(* IEC 61131-3 sources: MSMP/PLC_Station/Source/FB, 12 files *)

(* ---- FB_CANopenManager.st ---- *)
FUNCTION_BLOCK FB_CANopenManager
VAR_INPUT
 Enable:BOOL;
END_VAR
VAR_OUTPUT
 Ready:BOOL;
END_VAR
IF Enable THEN
 Ready:=TRUE;
ELSE
 Ready:=FALSE;
END_IF;
END_FUNCTION_BLOCK

(* ---- FB_ConnectionMonitor.st ---- *)
FUNCTION_BLOCK FB_ConnectionMonitor
VAR_INPUT Connected:BOOL; END_VAR
VAR_OUTPUT Alarm:BOOL; END_VAR
Alarm:=NOT Connected;
END_FUNCTION_BLOCK

(* ---- FB_DataAcquisition.st ---- *)
FUNCTION_BLOCK FB_DataAcquisition
VAR_INPUT
    Enable : BOOL;
END_VAR
VAR_OUTPUT
    Done : BOOL;
END_VAR

IF Enable THEN
    // TODO: Read 6 CANopen encoders
    Done := TRUE;
ELSE
    Done := FALSE;
END_IF;

END_FUNCTION_BLOCK

(* ---- FB_Diagnostics.st ---- *)
FUNCTION_BLOCK FB_Diagnostics
VAR_INPUT
 CAN_OK:BOOL;
 MODBUS_OK:BOOL;
END_VAR
VAR_OUTPUT
 SystemHealthy:BOOL;
END_VAR
SystemHealthy:=CAN_OK AND MODBUS_OK;
END_FUNCTION_BLOCK

(* ---- FB_Encoder.st ---- *)
FUNCTION_BLOCK FB_Encoder
VAR_INPUT
 PositionRaw:LREAL;
END_VAR
VAR_OUTPUT
 Position:LREAL;
END_VAR
Position:=PositionRaw;
END_FUNCTION_BLOCK

(* ---- FB_EncoderManager.st ---- *)
FUNCTION_BLOCK FB_EncoderManager
VAR_INPUT
    Enable : BOOL;
END_VAR
VAR_OUTPUT
    Healthy : BOOL;
END_VAR

Healthy := Enable;

// TODO:
// - Check encoder timeout
// - Check StatusWord
// - Validate Position

END_FUNCTION_BLOCK

(* ---- FB_Heartbeat.st ---- *)
FUNCTION_BLOCK FB_Heartbeat
VAR_IN_OUT Counter:DWORD; END_VAR
Counter:=Counter+1;
END_FUNCTION_BLOCK

(* ---- FB_ModbusMapping.st ---- *)
FUNCTION_BLOCK FB_ModbusMapping
VAR_INPUT
 Enable:BOOL;
END_VAR
VAR_OUTPUT
 Ready:BOOL;
END_VAR
Ready:=Enable;
// TODO: map runtime variables to Modbus registers
END_FUNCTION_BLOCK

(* ---- FB_ModbusSlave.st ---- *)
FUNCTION_BLOCK FB_ModbusSlave
VAR_INPUT
 Enable:BOOL;
END_VAR
VAR_OUTPUT
 Online:BOOL;
END_VAR
Online:=Enable;
END_FUNCTION_BLOCK

(* ---- FB_StationManager.st ---- *)
FUNCTION_BLOCK FB_StationManager
VAR_INPUT
    Enable : BOOL;
END_VAR
VAR_OUTPUT
    Online : BOOL;
END_VAR

Online := Enable;

// TODO:
// Update gStation runtime structure

END_FUNCTION_BLOCK

(* ---- FB_System.st ---- *)
FUNCTION_BLOCK FB_System
VAR_INPUT
    Enable : BOOL;
END_VAR
VAR_OUTPUT
    Ready : BOOL;
    Run : BOOL;
END_VAR
IF Enable THEN
    Ready:=TRUE;
    Run:=TRUE;
ELSE
    Ready:=FALSE;
    Run:=FALSE;
END_IF;
END_FUNCTION_BLOCK

(* ---- FB_Watchdog.st ---- *)
FUNCTION_BLOCK FB_Watchdog
VAR_IN_OUT Counter:DWORD; END_VAR
Counter:=Counter+1;
END_FUNCTION_BLOCK
